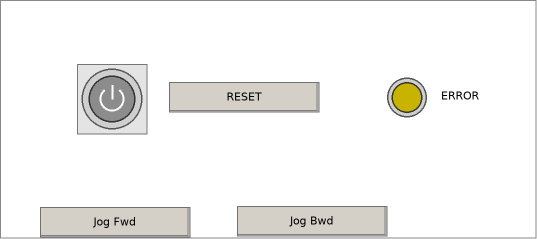
VISUALIZATION Visualization  // 537x239
    PowerSwitch (77,64 70x70), variable: MAIN.M1.bEnable, behaviour: TOGGLE, style: Switch-PowerSwitch-Gray
    Button (40,207 150x30), "Jog Fwd"
        tap MAIN.M1.bJogFwd
    Button (237,206 150x30), "Jog Bwd"
        tap MAIN.M1.bJogBwd
    Button (169,82 150x30), "RESET"
        tap MAIN.M1.bReset
    Lamp1 (384,73 46x49), variable: MAIN.M1.bError, style: Lamp-Lamp1-Yellow
    Label (385,81 150x30), "ERROR"
END_VISUALIZATION

(* stored: Version 1.1.0.1, ProductVersion 3.1.4018.5
   Visu Visualization: Id {2de5eae9-6b28-44ef-9999-f8c7f1eabd2c} *)
